FUNCTION_BLOCK FB_EPS
VAR_IN_OUT
    eps : DUT_EPS;
END_VAR
VAR_OUTPUT
END_VAR
VAR
END_VAR

METHOD setBit : BOOL
VAR_INPUT
    nBits : BYTE;
    bValue : BOOL;
END_VAR
VAR
    nMask : UDINT := 1;
    nBitValue : UDINT := 0;
END_VAR
nMask := SHL(nMask, nBits);
// Checking the VAR_IN_OUT reference, leave the current method in case of invalid reference
IF NOT __ISVALIDREF(eps) THEN
    RETURN;
END_IF

(* Access to VAR_IN_OUT reference (only if the reference was confirmed as valid before) *)
nBitValue := SHR((nMask AND eps.nFlags), nBits);

IF (TO_BOOL(nBitValue)) <> bValue THEN
    eps.nFlags := eps.nFlags XOR nMask;
END_IF

// Check if all values are true
IF eps.nFlags = 16#FFFFFFFF THEN
    eps.bEPS_OK := TRUE;
ELSE
    eps.bEPS_OK := FALSE;
END_IF
END_METHOD

METHOD setDescription : BOOL
VAR_INPUT
    desciption : STRING;
END_VAR

// Checking the VAR_IN_OUT reference, leave the current method in case of invalid reference
IF NOT __ISVALIDREF(eps) THEN
    RETURN;
END_IF

(* Access to VAR_IN_OUT reference (only if the reference was confirmed as valid before) *)
eps.sFlagDesc := desciption;
END_METHOD

METHOD setMessage : BOOL
VAR_INPUT
    message : STRING;
END_VAR
// Checking the VAR_IN_OUT reference, leave the current method in case of invalid reference
IF NOT __ISVALIDREF(eps) THEN
    RETURN;
END_IF
// Access to VAR_IN_OUT reference (only if the reference was confirmed as valid before)
eps.sMessage := message;
END_METHOD

END_FUNCTION_BLOCK

(* stored: Version 1.1.0.1
   POU FB_EPS: Id {0c78cf58-96ea-4c52-b0ca-64b7290d1ef9}, SpecialFunc None
   Method setBit: Id {243035d2-b889-46d7-b89e-610b76586068}
   Method setDescription: Id {84797ad0-c375-4675-8998-ec2e912fbbdd}
   Method setMessage: Id {50553b5a-8e8e-441f-8a78-c5cb5c67e718} *)
